INTERFACE I_HostInputPorts EXTENDS __SYSTEM.IQueryInterface

METHOD AddInputPort
VAR_INPUT
	InputPort : I_InputPort;
END_VAR
END_METHOD

METHOD PUBLIC TryGetInputPortByName : BOOL
VAR_INPUT
	Name : T_MAXSTRING;
	Destination : REFERENCE TO I_InputPort;
END_VAR
END_METHOD

END_INTERFACE

(* stored: Version 1.1.0.1, ProductVersion 3.1.4024.12
   Itf I_HostInputPorts: Id {20821798-bf3c-013b-3f9d-c61656a9dfcd}
   Method AddInputPort: Id {135eb44b-cbc4-0e2f-0792-05757aacdb77}
   Method TryGetInputPortByName: Id {a21ad5ef-ba3e-0598-3880-d9f06b97f2a5} *)
